ABB RobotStudio station: MarkerTool.rsstn

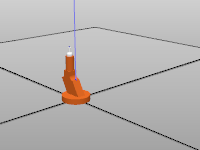
Station MarkerTool (saved by RobotStudio 20.4.9280.0)
Layout (positions relative to the parent item):
  - MarkerHolder [part]
  - Marker [part]
  - MarkerHolderTool [part]
